FUNCTION_BLOCK FB_HE_SolidAttenuatorSlotMock EXTENDS FB_FalliblePublicMock IMPLEMENTS I_HE_SolidAttenuatorSlot
VAR
    fbCenterPosition	: FB_QuantityLREALPublicMock;
    fbLength	: FB_QuantityLREALPublicMock;
    sMaterial	: T_MaxString;
    eState : E_HE_SolidAttenuatorSlotState;
    fbThickness : FB_QuantityLREALPublicMock;
    bHasSpecifiedFilter : BOOL;
    bIsEnabled : BOOL;
END_VAR


METHOD GetCenterPosition
VAR_INPUT
    CenterPosition	: I_QuantityLREALPublic;
END_VAR

CenterPosition.Copy(THIS^.fbCenterPosition);
END_METHOD


METHOD GetLength
VAR_INPUT
    Length	: I_QuantityLREALPublic;
END_VAR

Length.Copy(THIS^.fbLength);
END_METHOD


METHOD GetMaterial
VAR_IN_OUT
    Material	: T_MaxString;
END_VAR

Material := sMaterial;
END_METHOD


METHOD GetState : E_HE_SolidAttenuatorSlotState

GetState := THIS^.eState;
END_METHOD


METHOD GetThicknessAt
VAR_INPUT
    QueryPointInAxisCoordinates	: I_QuantityLREAL;
    Thickness	: I_QuantityLREALPublic;
END_VAR

Thickness.Copy(THIS^.fbThickness);
END_METHOD


METHOD HasSpecifiedFilter : BOOL
VAR_INPUT
    Filter	: I_HE_SolidAttenuatorFilter;
END_VAR

HasSpecifiedFilter := THIS^.bHasSpecifiedFilter;
END_METHOD


METHOD IsEnabled : BOOL

IsEnabled := THIS^.bIsEnabled;
END_METHOD


METHOD SetCenterPosition
VAR_INPUT
    Result	: I_QuantityLREAL;
END_VAR

THIS^.fbCenterPosition.Copy(Result);
END_METHOD


METHOD SetHasSpecifiedFilter
VAR_INPUT
    Result : BOOL;
END_VAR

THIS^.bHasSpecifiedFilter := Result;
END_METHOD


METHOD SetIsEnabled
VAR_INPUT
    Result : BOOL;
END_VAR

THIS^.bIsEnabled := Result;
END_METHOD


METHOD SetLength
VAR_INPUT
    Result : I_QuantityLREAL;
END_VAR

THIS^.fbLength.Copy(Result);
END_METHOD


METHOD SetMaterial
VAR_INPUT
    Result : T_MaxString;
END_VAR

THIS^.sMaterial := Result;
END_METHOD


METHOD SetState
VAR_INPUT
    Result : E_HE_SolidAttenuatorSlotState;
END_VAR

THIS^.eState := Result;
END_METHOD


METHOD SetThicknessAt
VAR_INPUT
    Result : I_QuantityLREAL;
END_VAR

THIS^.fbThickness.Copy(Result);
END_METHOD

END_FUNCTION_BLOCK

(* stored: Version 1.1.0.1
   POU FB_HE_SolidAttenuatorSlotMock: Id {86233f46-6d67-46da-9131-7c8c14641465}, SpecialFunc None
   Method GetCenterPosition: Id {999571a2-1076-4d04-b9ed-f0ef724e6017}
   Method GetLength: Id {ddc8856d-aa63-4639-9f78-92c225097a06}
   Method GetMaterial: Id {244ca2ad-1f6f-4891-ad66-5f826a45bb56}
   Method GetState: Id {1eb53064-c91b-48c7-bf3c-113e2a040a11}
   Method GetThicknessAt: Id {525137e3-4fff-4ff7-83a9-d4d1c127dbb6}
   Method HasSpecifiedFilter: Id {c0a19c00-f294-4851-9e32-afcdd6746d37}
   Method IsEnabled: Id {afc1f2ec-a317-4b12-9c0c-ca72cc57ca32}
   Method SetCenterPosition: Id {37911ff8-c0ea-455c-a59f-483856678859}
   Method SetHasSpecifiedFilter: Id {2dc5d4a7-3343-4cbe-8c16-ea506a80aeb3}
   Method SetIsEnabled: Id {24030b06-04c2-4c78-8dd1-2a93afb38da0}
   Method SetLength: Id {d1be8611-a05f-4160-9437-7a5bc8a7ae53}
   Method SetMaterial: Id {61fafa1a-1ffb-4772-9ed5-c6fb727b8155}
   Method SetState: Id {994bd3bf-5f1b-4829-9b46-2bdc15e01e3c}
   Method SetThicknessAt: Id {41c72cfc-e4e9-462b-a814-efa2a6367375} *)
